(* IEC 61131-3 sources: ironplc-benchmarks/benchmarks/minimal_repros, 49 files *)

(* ---- 29_function_block_instance.st ---- *)
(* P4013: Function block instantiation treated as duplicate POU declaration.

   Declaring a variable whose type is a FUNCTION_BLOCK causes P4013
   "POU declaration name is duplicated". This is standard IEC 61131-3
   behavior: you define a FUNCTION_BLOCK and then create instances of
   it as variables. IronPLC incorrectly treats the variable type
   reference as a second POU declaration.

   This is a regression in v0.184.0 (commit ceb2f6f8). It blocks all
   FUNCTION_BLOCK usage in oscat.st, which means all 294 testable
   functions fail in full mode.

   Error: P4013 - POU declaration name is duplicated
   OSCAT impact: full-mode blocker, all functions fail

   Compile with:
     ironplcc compile --dialect rusty benchmarks/minimal_repros/29_function_block_instance.st
*)

FUNCTION_BLOCK COUNTER
VAR
    count : INT;
END_VAR
    count := count + 1;
END_FUNCTION_BLOCK

PROGRAM main
VAR
    c : COUNTER;
END_VAR
    c();
END_PROGRAM

(* ---- 36_var_constant_array_bound.st ---- *)
(* P4030: VAR CONSTANT used as array bound not resolved.

   Using a VAR CONSTANT declared in the same FUNCTION_BLOCK as an
   array dimension bound fails with P4030 "Constant referenced in
   type parameter is not defined". The constant is defined after the
   array declaration in a separate VAR CONSTANT block.

   This pattern is used in OSCAT for configurable-size FIFO and STACK
   function blocks where the size is a local constant.

   Error: P4030 - Constant referenced in type parameter is not defined
   OSCAT impact: FIFO_16, FIFO_32, STACK_16, STACK_32 (4 function blocks)

   Compile with:
     ironplcc compile --dialect rusty benchmarks/minimal_repros/36_var_constant_array_bound.st
*)

FUNCTION_BLOCK MY_FIFO
VAR_INPUT
    din : DWORD;
END_VAR
VAR
    fifo : ARRAY[0..n] OF DWORD;
    idx : INT;
END_VAR
VAR CONSTANT
    n : INT := 16;
END_VAR
    fifo[idx] := din;
    idx := idx + 1;
    IF idx > n THEN idx := 0; END_IF;
END_FUNCTION_BLOCK

PROGRAM main
VAR
    f : MY_FIFO;
END_VAR
    f(din := DWORD#42);
END_PROGRAM

(* ---- 01_cross_function_call.st ---- *)
(* Category 1: Calling a function not defined in the compilation unit.
   compile.rs#L2116 — 49 OSCAT functions affected.
   e.g. CTRL_IN calls DEAD_ZONE, but DEAD_ZONE is not in the same file.
   NOTE: this works when both functions are in the same file. *)

FUNCTION OUTER : REAL
VAR_INPUT
    A : REAL;
    B : REAL;
    C : REAL;
END_VAR
    (* DEAD_ZONE is not defined here — triggers the error *)
    OUTER := DEAD_ZONE(A - B, C);
END_FUNCTION

PROGRAM main
VAR
    result : REAL;
END_VAR
    result := OUTER(A := 10.0, B := 3.0, C := 1.0);
END_PROGRAM

(* ---- 01b_string_func_in_function.st ---- *)
(* Category 1b: String stdlib function called from FUNCTION context.
   compile.rs#L2513 (LEN), #L2537 (FIND) — separate codegen paths.
   Works in PROGRAM, fails in FUNCTION.
   Affects COUNT_SUBSTRING, FSTRING_TO_WEEK, and other string-using functions. *)

FUNCTION MY_LEN : INT
VAR_INPUT
    S : STRING;
END_VAR
    MY_LEN := LEN(S);
END_FUNCTION

PROGRAM main
VAR
    result : INT;
END_VAR
    result := MY_LEN(S := 'Hello');
END_PROGRAM

(* ---- 01c_global_var_access.st ---- *)
(* Category 1c: Accessing an undefined global variable (dot notation).
   compile.rs#L3307 — 14 OSCAT functions affected.
   e.g. C_TO_K uses phys.T0, GAMMA uses math.PI2.
   Also: compile.rs#L3302 for global array indexing (math.FACTS[X]). *)

FUNCTION MY_FUNC : REAL
VAR_INPUT
    X : REAL;
END_VAR
    MY_FUNC := X - phys.T0;
END_FUNCTION

PROGRAM main
VAR
    result : REAL;
END_VAR
    result := MY_FUNC(X := 100.0);
END_PROGRAM

(* ---- 04_shl_with_function_arg.st ---- *)
(* Category 3: SHL/SHR with function call as first argument.
   Affects 15 OSCAT functions. *)

FUNCTION MY_SHIFT : WORD
VAR_INPUT
    B : BYTE;
END_VAR
    MY_SHIFT := SHL(BYTE_TO_WORD(B), 8);
END_FUNCTION

PROGRAM main
VAR
    result : WORD;
END_VAR
    result := MY_SHIFT(B := BYTE#16#AB);
END_PROGRAM

(* ---- 05_scientific_notation.st ---- *)
(* Category 4: Scientific notation in REAL literals (e.g. 2E-3).
   Part of 38 syntax errors. *)

FUNCTION APPROX : REAL
VAR_INPUT
    X : REAL;
END_VAR
    IF ABS(X) < 2E-3 THEN
        APPROX := X;
    ELSE
        APPROX := X * 1.5E+2;
    END_IF;
END_FUNCTION

PROGRAM main
VAR
    result : REAL;
END_VAR
    result := APPROX(X := 0.001);
END_PROGRAM

(* ---- 06_type_struct.st ---- *)
(* Category 5: TYPE STRUCT declarations.
   Part of 38 syntax errors. *)

TYPE MY_POINT :
STRUCT
    X : REAL;
    Y : REAL;
END_STRUCT
END_TYPE

PROGRAM main
VAR
    pt : MY_POINT;
END_VAR
    pt.X := 1.0;
    pt.Y := 2.0;
END_PROGRAM

(* ---- 07_array_indexing.st ---- *)
(* Category 7: Array indexing not implemented in codegen.
   Affects all OSCAT functions using arrays (ARRAY_* family, interpolation, etc.).
   Error: Not implemented at codegen/src/compile.rs#L3248 *)

PROGRAM main
VAR
    data : ARRAY[0..3] OF DINT;
    result : DINT;
END_VAR
    data[0] := 10;
    data[1] := 20;
    result := data[0] + data[1];
END_PROGRAM

(* ---- 09_ref_to.st ---- *)
(* Category 8: REF_TO / pointer dereference (Edition 3).
   Affects 45 OSCAT functions. *)

FUNCTION DEREF_ADD : REAL
VAR_INPUT
    P : REF_TO REAL;
    X : REAL;
END_VAR
    DEREF_ADD := P^ + X;
END_FUNCTION

PROGRAM main
VAR
    val : REAL := 10.0;
    result : REAL;
END_VAR
    result := DEREF_ADD(P := REF(val), X := 5.0);
END_PROGRAM

(* ---- 10_ltime.st ---- *)
(* Category 9: LTIME type (Edition 3).
   Affects 1 OSCAT function. *)

FUNCTION USE_LTIME : LTIME
VAR_INPUT
    X : LTIME;
END_VAR
    USE_LTIME := X;
END_FUNCTION

PROGRAM main
VAR
    result : LTIME;
END_VAR
    result := USE_LTIME(X := LTIME#100ms);
END_PROGRAM

(* ---- 11_unused_functions.st ---- *)
(* Demonstrates: multiple functions defined but only some are referenced.
   The compiler should compile this successfully by excluding unreferenced
   functions from codegen. Once supported, the compat test can include
   all of oscat.st and let the compiler tree-shake unused functions.

   Call graph:
     main -> OUTER -> INNER
     UNUSED_FUNC is defined but never called.
*)

FUNCTION INNER : REAL
VAR_INPUT
    X : REAL;
END_VAR
    INNER := X * 2.0;
END_FUNCTION

FUNCTION UNUSED_FUNC : REAL
VAR_INPUT
    X : REAL;
END_VAR
    (* This function is never called — compiler should skip it.
       It uses features that may not be implemented yet, but since
       it is unreferenced, compilation should still succeed. *)
    UNUSED_FUNC := SOME_UNDEFINED_FUNC(X) + 42.0;
END_FUNCTION

FUNCTION OUTER : REAL
VAR_INPUT
    A : REAL;
    B : REAL;
END_VAR
    OUTER := INNER(X := A) + B;
END_FUNCTION

PROGRAM main
VAR
    result : REAL;
END_VAR
    result := OUTER(A := 3.0, B := 1.0);
END_PROGRAM

(* ---- 12_terminal_error.st ---- *)
(* The compiler crashes trying to render the error diagnostic for this
   program. The actual error is hidden behind:
   "Failed writing to terminal: file missing"

   Root cause: accessing a global struct variable (e.g. setup.EXTENDED_ASCII)
   that is not defined in the compilation unit. The codegen hits a "not
   implemented" path, but the error renderer crashes before printing it.

   Affects 8 OSCAT functions: RDM2, FSTRING_TO_BYTE, FSTRING_TO_DWORD,
   ISC_ALPHA, ISC_LOWER, ISC_UPPER, DAYS_IN_YEAR, LEAP_OF_DATE.

   Note: unresolved function calls (compile.rs#L2430) render their error
   fine — only unresolved global variable access crashes the renderer. *)

FUNCTION TEST_FUNC : BOOL
VAR_INPUT
    X : BYTE;
END_VAR
    IF setup.EXTENDED_ASCII THEN
        TEST_FUNC := X > 64;
    ELSE
        TEST_FUNC := X > 96;
    END_IF;
END_FUNCTION

PROGRAM main
VAR
    result : BOOL;
END_VAR
    result := TEST_FUNC(X := BYTE#16#41);
END_PROGRAM

(* ---- 13_time_function_call.st ---- *)
(* TIME() used as a function call to read PLC system clock.
   IronPLC treats TIME as a type keyword and expects '#' for a literal,
   not '(' for a function call.

   Error: P0002 — Expected '#'. Found '('
   OSCAT functions affected: T_PLC_MS, T_PLC_US

   Compile with:
     ironplcc compile --allow-all --std-iec-61131-3 2013 -o /tmp/test.iplc benchmarks/minimal_repros/13_time_function_call.st
*)

FUNCTION T_PLC_MS : DWORD
VAR
    tx : TIME;
END_VAR
    tx := TIME();
    T_PLC_MS := TIME_TO_DWORD(tx);
END_FUNCTION

PROGRAM main
VAR
    result : DWORD;
END_VAR
    result := T_PLC_MS();
END_PROGRAM

(* ---- 14_missing_semicolon_end_if.st ---- *)
(* Missing semicolon after END_IF before END_FUNCTION.
   The --allow-missing-semicolon flag does not cover this case.

   Error: P0002 — Expected ';'. Found 'END_FUNCTION'
   OSCAT functions affected: SCALE_B

   Compile with:
     ironplcc compile --allow-all --std-iec-61131-3 2013 -o /tmp/test.iplc benchmarks/minimal_repros/14_missing_semicolon_end_if.st
*)

FUNCTION SCALE_B : REAL
VAR_INPUT
    X : BYTE;
    I_LO : BYTE;
    I_HI : BYTE;
    O_LO : REAL;
    O_HI : REAL;
END_VAR
    IF I_HI = I_LO THEN
        SCALE_B := O_LO;
    ELSE
        SCALE_B := O_HI;
    END_IF

END_FUNCTION

PROGRAM main
VAR
    result : REAL;
END_VAR
    result := SCALE_B(X := BYTE#1, I_LO := BYTE#0, I_HI := BYTE#10, O_LO := 0.0, O_HI := 100.0);
END_PROGRAM

(* ---- 15_end_struct_missing_semicolon.st ---- *)
(* Missing semicolon after END_STRUCT before END_TYPE.
   OSCAT consistently writes END_STRUCT without a trailing semicolon.

   Error: P0002 — Expected ';'. Found 'END_TYPE'
   OSCAT functions affected: CPOL, CSET, R2_SET, REAL_TO_FRAC,
     STATUS_TO_ESR, DT2_TO_SDT, DT_TO_SDT (via their TYPE dependencies)

   Compile with:
     ironplcc compile --allow-all --std-iec-61131-3 2013 -o /tmp/test.iplc benchmarks/minimal_repros/15_end_struct_missing_semicolon.st
*)

TYPE COMPLEX :
STRUCT
    re : REAL;
    im : REAL;
END_STRUCT
END_TYPE

FUNCTION CPOL_RE : REAL
VAR_INPUT
    L : REAL;
    A : REAL;
END_VAR
    CPOL_RE := L * COS(A);
END_FUNCTION

PROGRAM main
VAR
    result : REAL;
END_VAR
    result := CPOL_RE(L := 1.0, A := 0.0);
END_PROGRAM

(* ---- 16_var_temp.st ---- *)
(* VAR_TEMP block in FUNCTION declaration.
   IronPLC does not recognize VAR_TEMP as a valid variable section.
   Also blocks full-mode oscat.st parsing since FUNCTION_BLOCKs use VAR_TEMP.

   Error: P0002 — Found 'VAR_TEMP', expected identifier/statement
   OSCAT functions affected: REPLACE_UML (in FUNCTION),
     plus many FUNCTION_BLOCKs in full oscat.st

   Compile with:
     ironplcc compile --allow-all --std-iec-61131-3 2013 -o /tmp/test.iplc benchmarks/minimal_repros/16_var_temp.st
*)

FUNCTION MY_FUNC : INT
VAR_INPUT
    x : INT;
END_VAR
VAR_TEMP
    temp : INT;
END_VAR
    temp := x * 2;
    MY_FUNC := temp;
END_FUNCTION

PROGRAM main
VAR
    result : INT;
END_VAR
    result := MY_FUNC(x := 5);
END_PROGRAM

(* ---- 17_c_style_comment.st ---- *)
(* C-style block comment /* ... */ inside function body.
   IronPLC does not recognize /* */ comments, only (* *) comments.

   Error: P0002 — Found '/' unexpected
   OSCAT functions affected: LIST_RETRIEVE_LAST

   Compile with:
     ironplcc compile --allow-all --std-iec-61131-3 2013 -o /tmp/test.iplc benchmarks/minimal_repros/17_c_style_comment.st
*)

FUNCTION MY_FUNC : INT
VAR_INPUT
    x : INT;
END_VAR
    /* This is a C-style comment */
    MY_FUNC := x;
END_FUNCTION

PROGRAM main
VAR
    result : INT;
END_VAR
    result := MY_FUNC(x := 5);
END_PROGRAM

(* ---- 18_undefined_function_error_message.st ---- *)
(* Calling a function not defined in the compilation unit produces a
   misleading error message.

   Expected: a clear diagnostic like "function 'HELPER' is not defined"
   Actual: error[P9999]: Capability is not implemented (yet!)
           Not implemented at codegen/src/compile.rs#L2736

   This affects ~40 OSCAT functions when compiled in isolation (without
   the full oscat.st), since they call other OSCAT functions that aren't
   present in the compilation unit.

   Compile with:
     ironplcc compile --allow-all --std-iec-61131-3 2013 -o /tmp/test.iplc benchmarks/minimal_repros/18_undefined_function_error_message.st
*)

FUNCTION MY_FUNC : INT
VAR_INPUT
    x : INT;
END_VAR
    MY_FUNC := HELPER(x);
END_FUNCTION

PROGRAM main
VAR
    result : INT;
END_VAR
    result := MY_FUNC(x := 5);
END_PROGRAM

(* ---- 19_implicit_int_conversion.st ---- *)
(* P4026: Implicit integer type conversion not supported.

   IronPLC with --dialect rusty rejects passing an integer literal where
   a narrower integer type is expected. RuSTy and most PLC runtimes
   implicitly convert between integer types (e.g. DINT to INT).

   Error: P4026 — Function call argument type does not match parameter type
          (expected=INT, actual=DINT)
   OSCAT functions affected: 41 functions (BFT_TO_MS, BIT_LOAD_B, etc.)

   The fix should add an --allow-implicit-int-conversion flag (or include
   it in --dialect rusty) that permits implicit narrowing/widening
   conversions between integer types (SINT, INT, DINT, LINT and their
   unsigned variants) in function call arguments.

   Compile with:
     ironplcc compile --dialect rusty -o /tmp/test.iplc benchmarks/minimal_repros/19_implicit_int_conversion.st
*)

FUNCTION ADD_ONE : INT
VAR_INPUT
    x : INT;
END_VAR
    ADD_ONE := x + 1;
END_FUNCTION

PROGRAM main
VAR
    result : INT;
END_VAR
    (* 5 is inferred as DINT, but ADD_ONE expects INT *)
    result := ADD_ONE(x := 5);
END_PROGRAM

(* ---- 20_pointer_arithmetic.st ---- *)
(* P2033/P2035: Pointer arithmetic and comparison on REF_TO types.

   IronPLC rejects arithmetic (+, -) and ordering comparisons (<, >, <=, >=)
   on REF_TO types. RuSTy and OSCAT use pointer arithmetic extensively for
   efficient buffer and string manipulation.

   Errors:
     P2033 — Arithmetic operations are not allowed on reference types
     P2035 — Ordering comparison on reference types (only = and <> are allowed)
   OSCAT functions affected: 29 functions (CAPITALIZE, BIN_TO_BYTE, etc.)

   The fix should add an --allow-pointer-arithmetic flag (or include it
   in --dialect rusty) that permits arithmetic operations and ordering
   comparisons on REF_TO types, treating them as memory addresses.

   Compile with:
     ironplcc compile --dialect rusty -o /tmp/test.iplc benchmarks/minimal_repros/20_pointer_arithmetic.st
*)

FUNCTION FILL_ZEROS : BOOL
VAR_INPUT
    pt : REF_TO BYTE;
    size : INT;
END_VAR
VAR
    i : INT;
    end_ptr : REF_TO BYTE;
END_VAR
    end_ptr := pt + INT_TO_DWORD(size);    (* P2033: arithmetic on REF_TO *)
    WHILE pt < end_ptr DO                  (* P2035: comparison on REF_TO *)
        pt^ := 0;
        pt := pt + 1;                      (* P2033: arithmetic on REF_TO *)
    END_WHILE;
    FILL_ZEROS := TRUE;
END_FUNCTION

PROGRAM main
VAR
    result : BOOL;
END_VAR
    result := TRUE;
END_PROGRAM

(* ---- 21_ref_stack_variable.st ---- *)
(* P2029/P2032: REF() of stack-allocated variables and reference type punning.

   IronPLC rejects taking a reference to VAR_INPUT parameters in FUNCTION
   context (they are stack-allocated, so the reference would dangle after
   the function returns). It also rejects assigning a REF_TO of one type
   to a REF_TO of a different type.

   OSCAT uses this pattern for type punning — e.g. interpreting a REAL's
   bit pattern as a DWORD by taking REF(real_var) into a REF_TO DWORD.
   The reference never escapes the function, so it is safe in practice.

   Errors:
     P2029 — REF() of stack-allocated variable
     P2032 — Reference type mismatch in assignment
   OSCAT functions affected: 9 functions (CHK_REAL, DW_TO_REAL, REAL_TO_DW,
     CODE, FIND_CHAR, etc.)

   The fix should add an --allow-ref-stack-variables flag (or include it
   in --dialect rusty) that permits REF() on function-local and input
   variables, and an --allow-ref-type-punning flag that permits assigning
   between REF_TO types of different base types.

   Compile with:
     ironplcc compile --dialect rusty -o /tmp/test.iplc benchmarks/minimal_repros/21_ref_stack_variable.st
*)

FUNCTION CHK_REAL : BYTE
VAR_INPUT
    X : REAL;
END_VAR
VAR
    pt : REF_TO DWORD;
    tmp : DWORD;
END_VAR
    pt := REF(X);      (* P2029: REF of stack VAR_INPUT *)
                        (* P2032: REF_TO REAL assigned to REF_TO DWORD *)
    tmp := pt^;
    IF tmp < 16#7F800000 THEN
        CHK_REAL := 0;
    ELSE
        CHK_REAL := 16#80;
    END_IF;
END_FUNCTION

PROGRAM main
VAR
    result : BYTE;
END_VAR
    result := CHK_REAL(X := 1.0);
END_PROGRAM

(* ---- 22_undefined_global_variable.st ---- *)
(* P4007: Undefined global variables accessed via dotted notation.

   IronPLC rejects references to variables like math.PI, phys.T0, and
   setup.EXTENDED_ASCII because these global variable namespaces are not
   defined in the compilation unit. In OSCAT, these are defined as
   VAR_GLOBAL blocks that are expected to be linked from another file.

   Error: P4007 — Variable not defined before used
   OSCAT variables affected:
     math.PI, math.PI2, math.E, math.FACTS[] (13 functions)
     setup.EXTENDED_ASCII, setup.LANGUAGE (8 functions)
     LANGUAGE.DEFAULT, LANGUAGE.LMAX (6 functions)
     phys.T0, phys.C0, etc. (5 functions)

   The fix should add an --allow-undefined-globals flag (or include it in
   --dialect rusty) that treats unresolved dotted variable references as
   external globals rather than raising an error. This allows compilation
   units to reference globals defined elsewhere.

   Compile with:
     ironplcc compile --dialect rusty -o /tmp/test.iplc benchmarks/minimal_repros/22_undefined_global_variable.st
*)

FUNCTION C_TO_K : REAL
VAR_INPUT
    Celsius : REAL;
END_VAR
    C_TO_K := Celsius - phys.T0;     (* P4007: 'phys' not defined *)
END_FUNCTION

PROGRAM main
VAR
    result : REAL;
END_VAR
    result := C_TO_K(Celsius := 100.0);
END_PROGRAM

(* ---- 23_undefined_constant_type_param.st ---- *)
(* P4030: Constant referenced in type parameter is not defined.

   IronPLC with --allow-constant-type-params allows using constants in
   type parameters like STRING[MY_CONST], but the analyzer still requires
   the constant to be defined in the current compilation unit. OSCAT uses
   STRING[STRING_LENGTH] extensively, where STRING_LENGTH is a global
   constant defined elsewhere.

   Error: P4030 — Constant referenced in type parameter is not defined
   OSCAT functions affected: 9 functions (CLEAN, DEL_CHARS, FINDB,
     IS_CC, IS_NCC, REPLACE_CHARS, TRIM, TRIM1, TRIME)

   The fix should make --allow-constant-type-params (which is already
   included in --dialect rusty) also tolerate undefined constants in type
   parameters by using a default size, rather than raising an error.
   Alternatively, add a separate --allow-undefined-constant-type-params
   flag.

   Compile with:
     ironplcc compile --dialect rusty -o /tmp/test.iplc benchmarks/minimal_repros/23_undefined_constant_type_param.st
*)

FUNCTION MY_TRIM : STRING[STRING_LENGTH]
VAR_INPUT
    str : STRING[STRING_LENGTH];
END_VAR
    MY_TRIM := str;
END_FUNCTION

PROGRAM main
VAR
    result : STRING[255];
END_VAR
    result := MY_TRIM(str := 'hello');
END_PROGRAM

(* ---- 24_bool_int_initializer.st ---- *)
(* P4022: BOOL variable initialized with integer literal 0 or 1.

   IEC 61131-3 strictly requires TRUE/FALSE for BOOL, but initializing
   with 0 or 1 is a universal vendor extension supported by CoDeSys,
   TwinCAT, RuSTy, and virtually every PLC runtime.

   Error: P4022 — Variable initializer type is incompatible with
          declared type (variable=debug)
   OSCAT functions affected: T_PLC_MS, T_PLC_US

   The fix should include implicit integer-to-BOOL conversion in
   --dialect rusty, treating 0 as FALSE and non-zero as TRUE in
   variable initializers.

   Compile with:
     ironplcc compile --dialect rusty -o /tmp/test.iplc benchmarks/minimal_repros/24_bool_int_initializer.st
*)

FUNCTION MY_FUNC : DWORD
VAR CONSTANT
    debug : BOOL := 0;
END_VAR
    IF debug THEN
        MY_FUNC := 1;
    ELSE
        MY_FUNC := 0;
    END_IF;
END_FUNCTION

PROGRAM main
VAR
    result : DWORD;
END_VAR
    result := MY_FUNC();
END_PROGRAM

(* ---- 25_forward_ref_global_constant.st ---- *)
(* P9999: VAR_GLOBAL CONSTANT not handled in declaration toposort.

   Using a VAR_GLOBAL CONSTANT in STRING[MY_LENGTH] type parameters
   fails because the analyzer's toposort pass does not handle
   VAR_GLOBAL CONSTANT declarations.

   In OSCAT, STRING_LENGTH and LIST_LENGTH are defined as VAR_GLOBAL
   CONSTANT and used throughout oscat.st. This is the primary blocker
   for full-mode compilation — it fails regardless of whether the
   constant is declared before or after its use.

   Error: P9999 — Not implemented at analyzer/src/xform_toposort_declarations.rs#L535
   Also causes: P4030 when compiled in isolation without the constant
   OSCAT functions affected: 18+ functions (full-mode blocker)

   Compile with:
     ironplcc compile --dialect rusty -o /tmp/test.iplc benchmarks/minimal_repros/25_forward_ref_global_constant.st
*)

(* Case 1: constant declared AFTER use — matches oscat.st layout *)
FUNCTION MY_FUNC : STRING[MY_LENGTH]
VAR_INPUT
    str : STRING[MY_LENGTH];
END_VAR
    MY_FUNC := str;
END_FUNCTION

VAR_GLOBAL CONSTANT
    MY_LENGTH : INT := 250;
END_VAR

PROGRAM main
VAR
    result : STRING[250];
END_VAR
    result := MY_FUNC(str := 'hello');
END_PROGRAM

(* Note: if the above triggers a different error than P4030, try Case 2
   below which declares the constant BEFORE use but still fails.
   Uncomment Case 2 and comment out Case 1 to test. *)

(* Case 2: constant declared BEFORE use — still fails with P4030
VAR_GLOBAL CONSTANT
    MY_LENGTH : INT := 250;
END_VAR

FUNCTION MY_FUNC2 : STRING[MY_LENGTH]
VAR_INPUT
    str : STRING[MY_LENGTH];
END_VAR
    MY_FUNC2 := str;
END_FUNCTION

PROGRAM main
VAR
    result : STRING[250];
END_VAR
    result := MY_FUNC2(str := 'hello');
END_PROGRAM
*)

(* ---- 26_array_of_sized_string.st ---- *)
(* P9999: ARRAY OF STRING[N] not implemented in codegen.

   Declaring a variable or struct field as ARRAY[...] OF STRING[N]
   parses correctly but fails during code generation with P9999
   "Unsupported array element type".

   In OSCAT, the CONSTANTS_LANGUAGE struct uses patterns like:
     WEEKDAYS : ARRAY[1..3, 1..7] OF STRING[10] := [...]

   Error: P9999 - Unsupported array element type (codegen)
   OSCAT impact: TYPE CONSTANTS_LANGUAGE cannot be parsed, which
     blocks parsing all 370 functions when compiled together.

   Compile with:
     ironplcc compile --dialect rusty benchmarks/minimal_repros/26_array_of_sized_string.st
*)

(* Case 1: ARRAY OF STRING[N] in a PROGRAM variable *)
PROGRAM main
VAR
    names : ARRAY[1..3] OF STRING[10];
END_VAR
    names[1] := 'hello';
END_PROGRAM

(* Case 2: ARRAY OF STRING[N] in a TYPE STRUCT - matches oscat.st usage
TYPE MY_STRUCT :
STRUCT
    ITEMS : ARRAY[1..7] OF STRING[10] := ['Mon', 'Tue', 'Wed', 'Thu', 'Fri', 'Sat', 'Sun'];
END_STRUCT
END_TYPE

PROGRAM main2
VAR
    s : MY_STRUCT;
END_VAR
    s.ITEMS[1] := 'Monday';
END_PROGRAM
*)

(* ---- 27_struct_string_field.st ---- *)
(* P9999: STRING field in TYPE STRUCT not implemented in analyzer.

   Declaring a TYPE STRUCT with a STRING field (with or without a
   size specifier) causes "Not implemented" in the analyzer's
   intermediates/structure pass. The struct does not need to be
   referenced or used - its mere presence triggers the error.

   Structs with only numeric fields (INT, SINT, REAL, etc.) work fine.

   Error: P9999 - Not implemented at analyzer/src/intermediates/structure.rs#L276
   OSCAT types affected: CALENDAR, ESR_DATA, HOLIDAY_DATA
   OSCAT impact: blocks compilation of all 294 testable functions
     when compiled together with oscat.st (full mode), because the
     analyzer aborts on the struct definition before reaching any
     function.

   Compile with:
     ironplcc compile --dialect rusty benchmarks/minimal_repros/27_struct_string_field.st
*)

(* Case 1: STRING without size specifier *)
TYPE MY_DATA :
STRUCT
    NAME : STRING;
    VALUE : INT;
END_STRUCT
END_TYPE

PROGRAM main
VAR
    x : INT;
END_VAR
    x := 1;
END_PROGRAM

(* Case 2: STRING with size specifier - same error
TYPE MY_DATA2 :
STRUCT
    NAME : STRING[30];
    VALUE : INT;
END_STRUCT
END_TYPE

PROGRAM main2
VAR
    x : INT;
END_VAR
    x := 1;
END_PROGRAM
*)

(* ---- 28_sel_return_type_nested.st ---- *)
(* P4026: SEL/MUX return type inferred from selector, not value parameters.

   When the standard function SEL or MUX is used as a nested argument
   to another function call, its return type is incorrectly inferred
   from the selector parameter type, BOOL for SEL, ANY_INT for MUX,
   instead of from the value parameters.

   SEL[BOOL, REAL, REAL] should return REAL, but IronPLC infers BOOL.
   MUX[INT, REAL, REAL] should return REAL, but IronPLC infers ANY_INT.

   Direct assignment works correctly because the target type guides
   inference. Assigning to a variable first also works as a workaround.
   The bug only manifests when the result is passed directly as an
   argument to another function call.

   Error: P4026 - Function call argument type does not match parameter type
   OSCAT impact: blocks 294 functions in full mode because the METER
     function_block uses SEL nested in R2_ADD call, and any error
     anywhere blocks the entire compilation.

   Compile with:
     ironplcc compile --dialect rusty benchmarks/minimal_repros/28_sel_return_type_nested.st
*)

FUNCTION TAKES_REAL : REAL
VAR_INPUT
    Y : REAL;
END_VAR
    TAKES_REAL := Y;
END_FUNCTION

PROGRAM main
VAR
    r : REAL;
END_VAR
    r := TAKES_REAL(Y := SEL(TRUE, 0.0, 1.0));
END_PROGRAM

(* ---- 30_int_literal_to_real_param.st ---- *)
(* P4026: Integer literal passed to REAL parameter not implicitly converted.

   Passing an integer literal like 0 to a function parameter declared
   as REAL fails with P4026 type mismatch. The literal is typed as
   ANY_INT instead of being implicitly widened to REAL.

   Using 0.0 instead of 0 works as a workaround. RuSTy allows this
   implicit conversion.

   In OSCAT, the RDM function is called as RDM(0) where the parameter
   is declared as REAL. This single call in a FUNCTION_BLOCK blocks
   all 294 testable functions in full mode.

   Error: P4026 - Function call argument type does not match parameter type
   OSCAT impact: full-mode blocker, all 294 functions fail

   Compile with:
     ironplcc compile --dialect rusty benchmarks/minimal_repros/30_int_literal_to_real_param.st
*)

FUNCTION TAKES_REAL : REAL
VAR_INPUT
    x : REAL;
END_VAR
    TAKES_REAL := x;
END_FUNCTION

PROGRAM main
VAR
    r : REAL;
END_VAR
    r := TAKES_REAL(x := 0);
END_PROGRAM

(* ---- 31_time_date_conversions.st ---- *)
(* P4017: Time/date type conversion functions not declared.

   IEC 61131-3 defines type conversion functions between elementary
   types using the naming convention TYPE1_TO_TYPE2. IronPLC supports
   numeric conversions (INT_TO_REAL, etc.) but is missing conversions
   involving TIME, DATE, TOD, and DT types.

   These are used extensively in OSCAT for date/time arithmetic.
   In RuSTy, some are built-in and others are declared in stubs.st
   as EXTERNAL functions provided by the runtime.

   Error: P4017 - Function is not declared
   OSCAT functions affected: most date/time functions

   Compile with:
     ironplcc compile --dialect rusty benchmarks/minimal_repros/31_time_date_conversions.st
*)

PROGRAM main
VAR
    t : TIME := T#5s;
    d : DATE := D#2024-06-15;
    tod1 : TOD := TOD#12:30:00;
    dt1 : DT := DT#2024-06-15-12:30:00;
    dw : DWORD;
    ud : UDINT;
    di : DINT;
    r : REAL;
    i : INT;
    tm : TIME;
END_VAR
    dw := TIME_TO_DWORD(t);
    tm := DWORD_TO_TIME(dw);
    r := TIME_TO_REAL(t);
    di := TIME_TO_DINT(t);
    i := TIME_TO_INT(t);
    dw := DATE_TO_DWORD(d);
    ud := DATE_TO_UDINT(d);
    dw := TOD_TO_DWORD(tod1);
    dw := DT_TO_DWORD(dt1);
END_PROGRAM

(* ---- 32_sizeof.st ---- *)
(* P4017: SIZEOF operator not supported.

   SIZEOF returns the size in bytes of a variable or type. It is not
   part of IEC 61131-3 but is a CODESYS extension also supported by
   TwinCAT/Beckhoff and RuSTy. It requires compile-time knowledge
   of type sizes so it cannot be implemented as a user-defined function.

   In OSCAT, SIZEOF is used in buffer management functions that work
   with REF_TO pointers.

   Error: P4017 - Function is not declared
   OSCAT functions affected: buffer management functions (8 uses)

   Compile with:
     ironplcc compile --dialect rusty benchmarks/minimal_repros/32_sizeof.st
*)

PROGRAM main
VAR
    x : INT;
    y : DWORD;
    arr : ARRAY[1..10] OF INT;
    s : DINT;
END_VAR
    s := SIZEOF(x);
    s := SIZEOF(y);
    s := SIZEOF(arr);
END_PROGRAM

(* ---- 33_implicit_integer_widening.st ---- *)
(* P4026: Implicit type widening not supported in function arguments.

   IEC 61131-3 allows implicit widening conversions where the range
   and precision of the source type are preserved:
   - ANY_INT widening: SINT->INT->DINT->LINT, USINT->UINT->UDINT->ULINT
   - ANY_INT to ANY_REAL: SINT/INT/DINT->REAL, any integer->LREAL
   - ANY_REAL widening: REAL->LREAL
   - ANY_BIT widening: BOOL->BYTE->WORD->DWORD->LWORD

   Cross-family conversions (e.g. INT->WORD, BYTE->INT) and narrowing
   conversions (e.g. DINT->INT) should NOT be implicitly allowed.

   IronPLC currently rejects ALL implicit conversions in function
   arguments, including the valid widening ones.

   Error: P4026 - Function call argument type does not match parameter type
   OSCAT impact: full-mode blocker, all 294 functions fail

   Compile with:
     ironplcc compile --dialect rusty benchmarks/minimal_repros/33_implicit_integer_widening.st
*)

(* Target functions for each destination type *)
FUNCTION TAKES_INT : INT
VAR_INPUT x : INT; END_VAR TAKES_INT := x; END_FUNCTION

FUNCTION TAKES_DINT : DINT
VAR_INPUT x : DINT; END_VAR TAKES_DINT := x; END_FUNCTION

FUNCTION TAKES_LINT : LINT
VAR_INPUT x : LINT; END_VAR TAKES_LINT := x; END_FUNCTION

FUNCTION TAKES_UINT : UINT
VAR_INPUT x : UINT; END_VAR TAKES_UINT := x; END_FUNCTION

FUNCTION TAKES_UDINT : UDINT
VAR_INPUT x : UDINT; END_VAR TAKES_UDINT := x; END_FUNCTION

FUNCTION TAKES_ULINT : ULINT
VAR_INPUT x : ULINT; END_VAR TAKES_ULINT := x; END_FUNCTION

FUNCTION TAKES_REAL : REAL
VAR_INPUT x : REAL; END_VAR TAKES_REAL := x; END_FUNCTION

FUNCTION TAKES_LREAL : LREAL
VAR_INPUT x : LREAL; END_VAR TAKES_LREAL := x; END_FUNCTION

FUNCTION TAKES_WORD : WORD
VAR_INPUT x : WORD; END_VAR TAKES_WORD := x; END_FUNCTION

FUNCTION TAKES_DWORD : DWORD
VAR_INPUT x : DWORD; END_VAR TAKES_DWORD := x; END_FUNCTION

FUNCTION TAKES_LWORD : LWORD
VAR_INPUT x : LWORD; END_VAR TAKES_LWORD := x; END_FUNCTION

FUNCTION TAKES_BYTE : BYTE
VAR_INPUT x : BYTE; END_VAR TAKES_BYTE := x; END_FUNCTION

PROGRAM test_any_int_widening
VAR
    si : SINT := 1;
    i : INT := 1;
    di : DINT := 1;
    usi : USINT := 1;
    ui : UINT := 1;
    udi : UDINT := 1;
    ri : INT;
    rdi : DINT;
    rli : LINT;
    rui : UINT;
    rudi : UDINT;
    ruli : ULINT;
END_VAR
    (* Signed integer widening *)
    ri := TAKES_INT(x := si);       (* SINT -> INT *)
    rdi := TAKES_DINT(x := si);     (* SINT -> DINT *)
    rdi := TAKES_DINT(x := i);      (* INT -> DINT - the OSCAT blocker *)
    rli := TAKES_LINT(x := si);     (* SINT -> LINT *)
    rli := TAKES_LINT(x := i);      (* INT -> LINT *)
    rli := TAKES_LINT(x := di);     (* DINT -> LINT *)

    (* Unsigned integer widening *)
    rui := TAKES_UINT(x := usi);    (* USINT -> UINT *)
    rudi := TAKES_UDINT(x := usi);  (* USINT -> UDINT *)
    rudi := TAKES_UDINT(x := ui);   (* UINT -> UDINT *)
    ruli := TAKES_ULINT(x := usi);  (* USINT -> ULINT *)
    ruli := TAKES_ULINT(x := ui);   (* UINT -> ULINT *)
    ruli := TAKES_ULINT(x := udi);  (* UDINT -> ULINT *)
END_PROGRAM

PROGRAM test_int_to_real_widening
VAR
    si : SINT := 1;
    i : INT := 1;
    di : DINT := 1;
    r : REAL;
    lr : LREAL;
END_VAR
    (* Integer to REAL widening *)
    r := TAKES_REAL(x := si);       (* SINT -> REAL *)
    r := TAKES_REAL(x := i);        (* INT -> REAL *)
    r := TAKES_REAL(x := di);       (* DINT -> REAL *)

    (* REAL to LREAL widening *)
    lr := TAKES_LREAL(x := r);      (* REAL -> LREAL *)
END_PROGRAM

PROGRAM test_any_bit_widening
VAR
    bo : BOOL := TRUE;
    by : BYTE := BYTE#1;
    w : WORD := WORD#1;
    dw : DWORD := DWORD#1;
    rb : BYTE;
    rw : WORD;
    rdw : DWORD;
    rlw : LWORD;
END_VAR
    (* BOOL widening *)
    rb := TAKES_BYTE(x := bo);      (* BOOL -> BYTE *)
    rw := TAKES_WORD(x := bo);      (* BOOL -> WORD *)
    rdw := TAKES_DWORD(x := bo);    (* BOOL -> DWORD *)
    rlw := TAKES_LWORD(x := bo);    (* BOOL -> LWORD *)

    (* BYTE widening *)
    rw := TAKES_WORD(x := by);      (* BYTE -> WORD *)
    rdw := TAKES_DWORD(x := by);    (* BYTE -> DWORD *)
    rlw := TAKES_LWORD(x := by);    (* BYTE -> LWORD *)

    (* WORD widening *)
    rdw := TAKES_DWORD(x := w);     (* WORD -> DWORD *)
    rlw := TAKES_LWORD(x := w);     (* WORD -> LWORD *)

    (* DWORD widening *)
    rlw := TAKES_LWORD(x := dw);    (* DWORD -> LWORD *)
END_PROGRAM

(* ---- 33b_rejected_conversions.st ---- *)
(* These conversions should be REJECTED by the compiler.

   IEC 61131-3 does not allow implicit narrowing or cross-family
   conversions. Each case below should produce a compile error.
   IronPLC correctly rejects all of these today.

   This file is a negative test - it should NOT compile.

   Compile with:
     ironplcc compile --dialect rusty benchmarks/minimal_repros/33b_rejected_conversions.st
   Expected: compile errors on every conversion below
*)

FUNCTION TAKES_INT : INT
VAR_INPUT x : INT; END_VAR TAKES_INT := x; END_FUNCTION

FUNCTION TAKES_SINT : SINT
VAR_INPUT x : SINT; END_VAR TAKES_SINT := x; END_FUNCTION

FUNCTION TAKES_WORD : WORD
VAR_INPUT x : WORD; END_VAR TAKES_WORD := x; END_FUNCTION

FUNCTION TAKES_REAL : REAL
VAR_INPUT x : REAL; END_VAR TAKES_REAL := x; END_FUNCTION

FUNCTION TAKES_BOOL : BOOL
VAR_INPUT x : BOOL; END_VAR TAKES_BOOL := x; END_FUNCTION

PROGRAM test_narrowing_rejected
VAR
    di : DINT := 1;
    i : INT := 1;
    li : LINT := 1;
    lr : LREAL := 1.0;
    dw : DWORD := DWORD#1;
    ri : INT;
    rsi : SINT;
    rr : REAL;
    rw : WORD;
END_VAR
    (* Narrowing - should all fail *)
    ri := TAKES_INT(x := di);       (* DINT -> INT: narrowing *)
    rsi := TAKES_SINT(x := i);      (* INT -> SINT: narrowing *)
    ri := TAKES_INT(x := li);       (* LINT -> INT: narrowing *)
    rr := TAKES_REAL(x := lr);      (* LREAL -> REAL: narrowing *)
    rw := TAKES_WORD(x := dw);      (* DWORD -> WORD: narrowing *)
END_PROGRAM

PROGRAM test_cross_family_rejected
VAR
    i : INT := 1;
    w : WORD := WORD#1;
    by : BYTE := BYTE#1;
    bo : BOOL := TRUE;
    ri : INT;
    rw : WORD;
    rb : BOOL;
END_VAR
    (* Cross-family - should all fail *)
    rw := TAKES_WORD(x := i);       (* INT -> WORD: num to bit *)
    ri := TAKES_INT(x := w);        (* WORD -> INT: bit to num *)
    ri := TAKES_INT(x := by);       (* BYTE -> INT: bit to num *)
    ri := TAKES_INT(x := bo);       (* BOOL -> INT: bit to num *)
    rb := TAKES_BOOL(x := i);       (* INT -> BOOL: num to bit *)
END_PROGRAM

(* ---- 34_system_up_time_global.st ---- *)
(* P4007: __SYSTEM_UP_TIME global variable not exposed.

   The rusty dialect lists --allow-system-uptime-global which should
   expose __SYSTEM_UP_TIME and __SYSTEM_UP_LTIME as implicit VAR_GLOBALs
   providing runtime monotonic uptime. However, the variable is not
   actually available and produces P4007 "Variable not defined".

   Error: P4007 - Variable not defined before used
   OSCAT impact: needed to implement TIME() function in compat library

   Compile with:
     ironplcc compile --dialect rusty benchmarks/minimal_repros/34_system_up_time_global.st
*)

PROGRAM main
VAR
    t : TIME;
END_VAR
    t := __SYSTEM_UP_TIME;
END_PROGRAM

(* ---- 35_declare_function_time.st ---- *)
(* P0002: Cannot declare a function named TIME.

   The rusty dialect includes --allow-time-as-function-name which
   allows calling TIME() as a function. However, declaring
   FUNCTION TIME is rejected by the parser because TIME is still
   treated as a keyword in the declaration context.

   This prevents creating a user-defined TIME function in a
   compatibility library to wrap __SYSTEM_UP_TIME.

   Error: P0002 - Syntax error (parser rejects TIME as function name)
   OSCAT impact: 2 calls to TIME() in OSCAT, needed for compat library

   Compile with:
     ironplcc compile --dialect rusty benchmarks/minimal_repros/35_declare_function_time.st
*)

FUNCTION TIME : TIME
    TIME := T#0s;
END_FUNCTION

PROGRAM main
VAR
    t : TIME;
END_VAR
    t := TIME();
END_PROGRAM

(* ---- 37_global_var_in_function.st ---- *)
(* P4007: VAR_GLOBAL not accessible from FUNCTION or FUNCTION_BLOCK.

   Variables declared in VAR_GLOBAL blocks cannot be read from
   FUNCTION or FUNCTION_BLOCK bodies. They work in PROGRAM context.

   In OSCAT, global constants STRING_LENGTH, LIST_LENGTH, and struct
   globals like phys.T0, math.FACTS are used from functions.

   Error: P4007 - Variable not defined before used
   OSCAT impact: 9 functions (DWORD_TO_STRF, FILL, FIX, LIST_ADD,
     LIST_CLEAN, LIST_INSERT, LIST_RETRIEVE, LIST_RETRIEVE_LAST,
     REPLACE_UML) plus C_TO_K etc via phys/math globals

   Compile with:
     ironplcc compile --dialect rusty benchmarks/minimal_repros/37_global_var_in_function.st
*)

VAR_GLOBAL CONSTANT
    MY_CONST : INT := 100;
END_VAR

FUNCTION USE_GLOBAL : INT
    USE_GLOBAL := MY_CONST;
END_FUNCTION

PROGRAM main
VAR
    r : INT;
END_VAR
    r := USE_GLOBAL();
END_PROGRAM

(* ---- 38_global_struct_field_access.st ---- *)
(* P9999: Accessing field of a global struct variable in a FUNCTION.

   Functions that reference fields of global struct variables like
   phys.T0 or math.FACTS[X] fail in codegen. The struct field
   access on a global is not implemented.

   Error: P9999 - Not implemented at codegen
   OSCAT impact: 36 functions (C_TO_K, DEG_TO_DIR, FACT, BETA, etc.)

   Compile with:
     ironplcc compile --dialect rusty benchmarks/minimal_repros/38_global_struct_field_access.st
*)

TYPE MY_CONSTANTS :
STRUCT
    PI : REAL := 3.14159;
    T0 : REAL := 273.15;
END_STRUCT
END_TYPE

VAR_GLOBAL CONSTANT
    phys : MY_CONSTANTS;
END_VAR

FUNCTION CELSIUS_TO_KELVIN : REAL
VAR_INPUT
    c : REAL;
END_VAR
    CELSIUS_TO_KELVIN := c - phys.T0;
END_FUNCTION

PROGRAM main
VAR
    r : REAL;
END_VAR
    r := CELSIUS_TO_KELVIN(c := 100.0);
END_PROGRAM

(* ---- 39_deref_array_subscript.st ---- *)
(* P9999: Array subscript on dereferenced REF_TO ARRAY OF BYTE.

   Expressions like pt^[i] where pt is REF_TO ARRAY[..] OF BYTE
   fail during code generation. This pattern is used in OSCAT for
   byte-level string manipulation via REF(str) cast to byte array.

   REF_TO ARRAY OF REAL works, but BYTE does not.

   Error: P9999 - Not implemented at codegen/src/compile_array.rs#L138
   OSCAT impact: 8 functions (LIST_GET, LIST_LEN, FIND_CHAR,
     FIND_CTRL, FIND_NONUM, FIND_NUM, FLOAT_TO_REAL, MIRROR)

   Compile with:
     ironplcc compile --dialect rusty benchmarks/minimal_repros/39_deref_array_subscript.st
*)

FUNCTION GET_BYTE : BYTE
VAR_INPUT
    pt : REF_TO ARRAY[1..255] OF BYTE;
    i : INT;
END_VAR
    GET_BYTE := pt^[i];
END_FUNCTION

PROGRAM main
VAR
    arr : ARRAY[1..255] OF BYTE;
    r : BYTE;
END_VAR
    arr[1] := BYTE#42;
    r := GET_BYTE(pt := REF(arr), i := 1);
END_PROGRAM

(* ---- 40_global_array_subscript.st ---- *)
(* P9999: Array subscript on global struct member not implemented.

   Accessing an array field of a global struct like math.FACTS[X]
   fails in codegen. This combines global struct access with array
   subscripting.

   Error: P9999 - Not implemented at codegen/src/compile_array.rs#L155
   OSCAT impact: 6 functions (FACT, DATE_ADD, DAY_OF_MONTH,
     DT2_TO_SDT, DT_TO_SDT, MONTH_BEGIN)

   Compile with:
     ironplcc compile --dialect rusty benchmarks/minimal_repros/40_global_array_subscript.st
*)

TYPE MY_MATH :
STRUCT
    FACTS : ARRAY[0..10] OF REAL;
END_STRUCT
END_TYPE

VAR_GLOBAL CONSTANT
    math : MY_MATH;
END_VAR

FUNCTION LOOKUP : REAL
VAR_INPUT
    x : INT;
END_VAR
    LOOKUP := math.FACTS[x];
END_FUNCTION

PROGRAM main
VAR
    r : REAL;
END_VAR
    r := LOOKUP(x := 5);
END_PROGRAM

(* ---- 41_nested_function_call_in_function_arg.st ---- *)
(* P9999: Nested stdlib function call as argument to another stdlib function.

   Calling a standard string function like FIND where one argument
   is itself a function call (e.g. FIND(str, MID(s, 1, n))) fails
   in codegen. The nested function call result is not handled as
   an argument.

   Error: P9999 - Not implemented at codegen/src/compile.rs#L4055
   OSCAT impact: 7 functions (CLEAN, DEL_CHARS, FSTRING_TO_BYTE,
     FSTRING_TO_DWORD, IS_CC, IS_NCC, REPLACE_CHARS)

   Compile with:
     ironplcc compile --dialect rusty benchmarks/minimal_repros/41_nested_function_call_in_function_arg.st
*)

FUNCTION MY_SEARCH : INT
VAR_INPUT
    haystack : STRING[255];
    needle : STRING[255];
    maxlen : INT;
END_VAR
    MY_SEARCH := FIND(haystack, MID(needle, 1, maxlen));
END_FUNCTION

PROGRAM main
VAR
    r : INT;
END_VAR
    r := MY_SEARCH(haystack := 'hello world', needle := 'world', maxlen := 3);
END_PROGRAM

(* ---- 42_string_comparison_operators.st ---- *)
(* P9999: Global struct field access blocks BYTE comparison codegen.

   Functions like ISC_ALPHA that compare BYTE values with integer
   literals (in > 64 AND in < 91) fail because they also access
   global struct fields like setup.EXTENDED_ASCII. The error
   appears at :1:1 because the global access fails before reaching
   the comparison code.

   This is the same root cause as #38 (global struct field access
   in functions) but manifests in character classification functions.

   Error: P9999 - Not implemented at codegen/src/compile.rs#L2072
   OSCAT impact: 7 functions (IS_ALNUM, IS_ALPHA, IS_LOWER,
     IS_UPPER, ISC_ALPHA, ISC_LOWER, ISC_UPPER)

   Compile with:
     ironplcc compile --dialect rusty benchmarks/minimal_repros/42_string_comparison_operators.st
*)

TYPE SETUP_DATA :
STRUCT
    EXTENDED_ASCII : BOOL := TRUE;
END_STRUCT
END_TYPE

VAR_GLOBAL CONSTANT
    setup : SETUP_DATA;
END_VAR

FUNCTION ISC_ALPHA : BOOL
VAR_INPUT
    in : BYTE;
END_VAR
    IF setup.EXTENDED_ASCII THEN
        ISC_ALPHA := (in > 64 AND in < 91) OR (in > 96 AND in < 123);
    ELSE
        ISC_ALPHA := (in > 64 AND in < 91) OR (in > 96 AND in < 123);
    END_IF;
END_FUNCTION

PROGRAM main
VAR
    r : BOOL;
END_VAR
    r := ISC_ALPHA(in := BYTE#72);
END_PROGRAM

(* ---- 43_string_char_index.st ---- *)
(* P9999: String character indexing via FIND/MID patterns not implemented.

   Functions that use FINDB-style byte-level string searching with
   comparison operators on individual characters fail in codegen.
   This covers patterns like comparing characters extracted from
   strings against character ranges.

   Error: P9999 - Not implemented at codegen/src/compile.rs#L2074
   OSCAT impact: 6 functions (CHARCODE, FINDB, FINDB_NONUM,
     FINDP, REPLACE_ALL, TRIM1, TRIME)

   Compile with:
     ironplcc compile --dialect rusty benchmarks/minimal_repros/43_string_char_index.st
*)

FUNCTION FIND_BACKWARDS : INT
VAR_INPUT
    str : STRING[255];
    ch : STRING[1];
END_VAR
VAR
    i : INT;
    c : STRING[1];
END_VAR
    FOR i := LEN(str) TO 1 BY -1 DO
        c := MID(str, 1, i);
        IF c = ch THEN
            FIND_BACKWARDS := i;
            RETURN;
        END_IF;
    END_FOR;
    FIND_BACKWARDS := 0;
END_FUNCTION

PROGRAM main
VAR
    r : INT;
END_VAR
    r := FIND_BACKWARDS(str := 'hello', ch := 'l');
END_PROGRAM

(* ---- 44_constant_overflow.st ---- *)
(* P2026: Constant value overflows target type.

   A DWORD constant with value 4294967292 (0xFFFFFFFC, which is -4
   in signed 32-bit) triggers an overflow error. This value fits in
   DWORD (unsigned 32-bit) but the compiler may be treating it as
   signed.

   Error: P2026 - Constant value overflows the target type
   OSCAT impact: 1 function (LAMBERT_W)

   Compile with:
     ironplcc compile --dialect rusty benchmarks/minimal_repros/44_constant_overflow.st
*)

FUNCTION MY_FUNC : REAL
VAR
    mask : DWORD := 4294967292;
END_VAR
    MY_FUNC := 0.0;
END_FUNCTION

PROGRAM main
VAR
    r : REAL;
END_VAR
    r := MY_FUNC();
END_PROGRAM

(* ---- 45_global_struct_with_string.st ---- *)
(* P9999: Global struct variable with STRING field not supported in codegen.

   Instantiating a TYPE STRUCT that contains a STRING field as a
   VAR_GLOBAL variable fails with "Structure contains unsupported
   field types (STRING, WSTRING, or FunctionBlock)".

   The struct definition itself is accepted. Using the struct as a
   local variable in a PROGRAM also works. Only VAR_GLOBAL
   instantiation fails.

   In OSCAT, the global variables LANGUAGE (CONSTANTS_LANGUAGE) and
   SETUP (CONSTANTS_SETUP) contain STRING fields, and their presence
   in VAR_GLOBAL blocks all 294 functions in full mode.

   Error: P9999 - Structure contains unsupported field types
   OSCAT impact: full-mode blocker, all 294 functions fail

   Compile with:
     ironplcc compile --dialect rusty benchmarks/minimal_repros/45_global_struct_with_string.st
*)

TYPE MY_DATA :
STRUCT
    NAME : STRING[30];
    VALUE : INT;
END_STRUCT
END_TYPE

VAR_GLOBAL
    data1 : MY_DATA;
END_VAR

PROGRAM main
VAR
    x : INT;
END_VAR
    x := 1;
END_PROGRAM

(* ---- 46_function_return_struct_field.st ---- *)
(* P9999: Assigning STRING or ARRAY field on function return struct.

   When a function returns a struct, assigning to a STRING field or
   an ARRAY element of the return value fails in codegen. Simple
   numeric field assignments (MAKE_ESR.typ := 1) work fine.

   Error: P9999 - Not implemented at codegen
   OSCAT impact: 1 function (STATUS_TO_ESR)

   Compile with:
     ironplcc compile --dialect rusty benchmarks/minimal_repros/46_function_return_struct_field.st
*)

TYPE MY_DATA :
STRUCT
    TYP : BYTE;
    NAME : STRING[10];
    VALUES : ARRAY[0..3] OF BYTE;
END_STRUCT
END_TYPE

FUNCTION MAKE_DATA : MY_DATA
VAR_INPUT
    t : BYTE;
    n : STRING[10];
END_VAR
    MAKE_DATA.TYP := t;
    MAKE_DATA.NAME := n;
    MAKE_DATA.VALUES[0] := t;
END_FUNCTION

PROGRAM main
VAR
    d : MY_DATA;
END_VAR
    d := MAKE_DATA(t := BYTE#1, n := 'test');
END_PROGRAM

(* ---- 47_global_multidim_array_subscript.st ---- *)
(* P9999: Multi-dimensional array subscript on global struct field.

   Accessing a multi-dimensional array field of a global struct
   variable like language.WEEKDAYS[ly, wday] fails in codegen.

   Error: P9999 - Not implemented at codegen
   OSCAT impact: 2 functions (MONTH_TO_STRING, WEEKDAY_TO_STRING)

   Compile with:
     ironplcc compile --dialect rusty benchmarks/minimal_repros/47_global_multidim_array_subscript.st
*)

TYPE MY_LANG :
STRUCT
    NAMES : ARRAY[1..2, 1..3] OF STRING[10] := [
        'Mon', 'Tue', 'Wed',
        'Mo', 'Di', 'Mi'];
END_STRUCT
END_TYPE

VAR_GLOBAL
    lang : MY_LANG;
END_VAR

FUNCTION GET_NAME : STRING[10]
VAR_INPUT
    row : INT;
    col : INT;
END_VAR
    GET_NAME := lang.NAMES[row, col];
END_FUNCTION

PROGRAM main
VAR
    s : STRING[10];
END_VAR
    s := GET_NAME(row := 1, col := 1);
END_PROGRAM

(* ---- 51_dword_constant_overflow.st ---- *)
(* P2026: DWORD hex literal overflows when used in comparison expression.

   Using a large DWORD hex literal like 16#FFFF_FFFC in both an
   assignment and an IF comparison causes P2026 "Constant value
   overflows the target type". The value 4294967292 fits in DWORD
   (unsigned 32-bit) but the codegen appears to evaluate it as
   signed during comparison.

   Using the literal once (in assignment only) works fine.

   Error: P2026 - Constant value overflows the target type
   OSCAT impact: 1 function (LAMBERT_W)

   Compile with:
     ironplcc compile --dialect rusty benchmarks/minimal_repros/51_dword_constant_overflow.st
*)

FUNCTION GET_DW : DWORD
VAR_INPUT x : REAL; END_VAR
    GET_DW := REAL_TO_DWORD(x);
END_FUNCTION

FUNCTION TEST_FUNC : REAL
VAR_INPUT x : REAL; END_VAR
VAR
    w : REAL := 1.0;
    last : DWORD;
END_VAR
    last := GET_DW(w) AND 16#FFFF_FFFC;
    IF (GET_DW(w) AND 16#FFFF_FFFC) = last THEN
        TEST_FUNC := w;
    END_IF;
END_FUNCTION

PROGRAM main
VAR r : REAL; END_VAR
    r := TEST_FUNC(x := 1.0);
END_PROGRAM

(* ---- 53_string_compare_in_if.st ---- *)
(* P9999: STRING comparison as IF condition not implemented in codegen.

   Using a STRING equality (or other comparison) as the condition of
   an IF statement triggers compile_expr.rs#L34. Direct assignment of
   the comparison result (CMP := a = b) works fine.

   This affects all functions that conditionally branch on string
   equality, which is a very common pattern.

   Suspected root cause (per compiler dev): "STRING outside the
   dedicated string-compare path".

   Error: P9999 - Not implemented at codegen/src/compile_expr.rs#L34
   OSCAT impact: 14 functions including DIR_TO_DEG (compares
     language.DIRS[ly,i] = DIR), CHARCODE, FINDB, REPLACE_ALL,
     TRIM1, TRIME, FSTRING_TO_*, EXEC

   Compile with:
     ironplcc compile --dialect rusty benchmarks/minimal_repros/52_string_compare_in_if.st
*)

FUNCTION COMPARE_STRINGS : BOOL
VAR_INPUT
    a : STRING[10];
    b : STRING[10];
END_VAR
    IF a = b THEN
        COMPARE_STRINGS := TRUE;
    ELSE
        COMPARE_STRINGS := FALSE;
    END_IF;
END_FUNCTION

PROGRAM main
VAR
    r : BOOL;
END_VAR
    r := COMPARE_STRINGS(a := 'hello', b := 'world');
END_PROGRAM
